FUNCTION_BLOCK TM_DO32 (* Composite Function Block Type *)
  (* Standard: 61499-2 *)
  (* Version 0.0, 21/08/2026, template *)
  PACKAGE Hidryco.HidrycoLib;
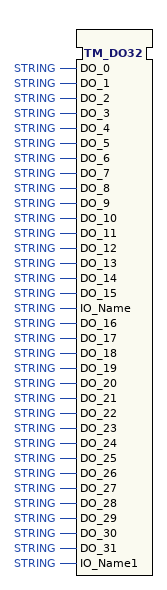
  VAR_INPUT
    DO_0 : STRING;
    DO_1 : STRING;
    DO_2 : STRING;
    DO_3 : STRING;
    DO_4 : STRING;
    DO_5 : STRING;
    DO_6 : STRING;
    DO_7 : STRING;
    DO_8 : STRING;
    DO_9 : STRING;
    DO_10 : STRING;
    DO_11 : STRING;
    DO_12 : STRING;
    DO_13 : STRING;
    DO_14 : STRING;
    DO_15 : STRING;
    IO_Name : STRING;
    DO_16 : STRING;
    DO_17 : STRING;
    DO_18 : STRING;
    DO_19 : STRING;
    DO_20 : STRING;
    DO_21 : STRING;
    DO_22 : STRING;
    DO_23 : STRING;
    DO_24 : STRING;
    DO_25 : STRING;
    DO_26 : STRING;
    DO_27 : STRING;
    DO_28 : STRING;
    DO_29 : STRING;
    DO_30 : STRING;
    DO_31 : STRING;
    IO_Name1 : STRING;
  END_VAR
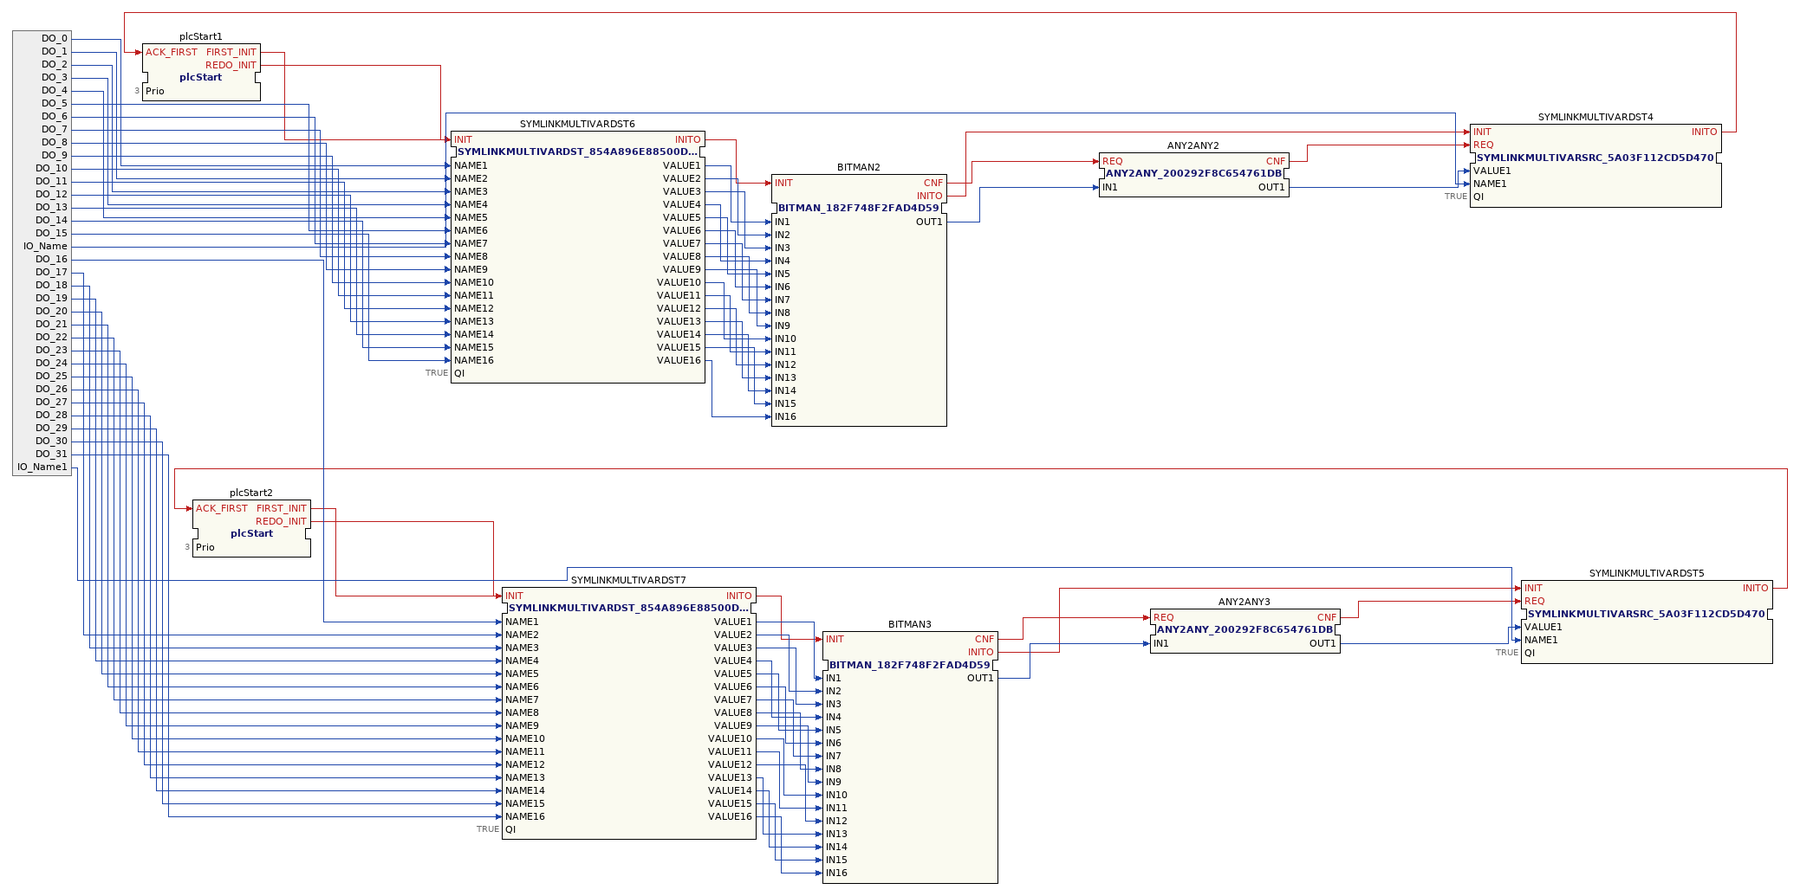
  FBS
    BITMAN2 : BITMAN_182F748F2FAD4D59; {SET_ATTRIBUTE(Configuration.GenericFBType.InterfaceParams, Runtime.Standard#CNTIN:=16;CNTOUT:=1;IN${CNTIN$}:BOOL,BOOL,BOOL,BOOL,BOOL,BOOL,BOOL,BOOL,BOOL,BOOL,BOOL,BOOL,BOOL,BOOL,BOOL,BOOL;OUT${CNTOUT$}:WORD)}
    ANY2ANY2 : ANY2ANY_200292F8C654761DB; {SET_ATTRIBUTE(Configuration.GenericFBType.InterfaceParams, Runtime.Standard#CNT:=1;IN${CNT$}:WORD;OUT${CNT$}:INT)}
    SYMLINKMULTIVARDST4 : SYMLINKMULTIVARSRC_5A03F112CD5D470(QI := TRUE); {SET_ATTRIBUTE(Configuration.GenericFBType.InterfaceParams, Runtime.System#I:=1;VALUE${I$}:INT)}
    SYMLINKMULTIVARDST6 : SYMLINKMULTIVARDST_854A896E88500D19(QI := TRUE); {SET_ATTRIBUTE(Configuration.GenericFBType.InterfaceParams, Runtime.System#I:=16;VALUE${I$}:BOOL,BOOL,BOOL,BOOL,BOOL,BOOL,BOOL,BOOL,BOOL,BOOL,BOOL,BOOL,BOOL,BOOL,BOOL,BOOL)}
    plcStart1 : plcStart(Prio := 3);
    BITMAN3 : BITMAN_182F748F2FAD4D59; {SET_ATTRIBUTE(Configuration.GenericFBType.InterfaceParams, Runtime.Standard#CNTIN:=16;CNTOUT:=1;IN${CNTIN$}:BOOL,BOOL,BOOL,BOOL,BOOL,BOOL,BOOL,BOOL,BOOL,BOOL,BOOL,BOOL,BOOL,BOOL,BOOL,BOOL;OUT${CNTOUT$}:WORD)}
    ANY2ANY3 : ANY2ANY_200292F8C654761DB; {SET_ATTRIBUTE(Configuration.GenericFBType.InterfaceParams, Runtime.Standard#CNT:=1;IN${CNT$}:WORD;OUT${CNT$}:INT)}
    SYMLINKMULTIVARDST5 : SYMLINKMULTIVARSRC_5A03F112CD5D470(QI := TRUE); {SET_ATTRIBUTE(Configuration.GenericFBType.InterfaceParams, Runtime.System#I:=1;VALUE${I$}:INT)}
    SYMLINKMULTIVARDST7 : SYMLINKMULTIVARDST_854A896E88500D19(QI := TRUE); {SET_ATTRIBUTE(Configuration.GenericFBType.InterfaceParams, Runtime.System#I:=16;VALUE${I$}:BOOL,BOOL,BOOL,BOOL,BOOL,BOOL,BOOL,BOOL,BOOL,BOOL,BOOL,BOOL,BOOL,BOOL,BOOL,BOOL)}
    plcStart2 : plcStart(Prio := 3);
  END_FBS
  EVENT_CONNECTIONS
    BITMAN2.CNF TO ANY2ANY2.REQ;
    BITMAN2.INITO TO SYMLINKMULTIVARDST4.INIT;
    ANY2ANY2.CNF TO SYMLINKMULTIVARDST4.REQ;
    SYMLINKMULTIVARDST6.INITO TO BITMAN2.INIT;
    plcStart1.FIRST_INIT TO SYMLINKMULTIVARDST6.INIT;
    plcStart1.REDO_INIT TO SYMLINKMULTIVARDST6.INIT;
    SYMLINKMULTIVARDST4.INITO TO plcStart1.ACK_FIRST;
    BITMAN3.CNF TO ANY2ANY3.REQ;
    BITMAN3.INITO TO SYMLINKMULTIVARDST5.INIT;
    ANY2ANY3.CNF TO SYMLINKMULTIVARDST5.REQ;
    SYMLINKMULTIVARDST7.INITO TO BITMAN3.INIT;
    plcStart2.FIRST_INIT TO SYMLINKMULTIVARDST7.INIT;
    plcStart2.REDO_INIT TO SYMLINKMULTIVARDST7.INIT;
    SYMLINKMULTIVARDST5.INITO TO plcStart2.ACK_FIRST;
  END_CONNECTIONS
  DATA_CONNECTIONS
    BITMAN2.OUT1 TO ANY2ANY2.IN1;
    ANY2ANY2.OUT1 TO SYMLINKMULTIVARDST4.VALUE1;
    SYMLINKMULTIVARDST6.VALUE1 TO BITMAN2.IN1;
    SYMLINKMULTIVARDST6.VALUE2 TO BITMAN2.IN2;
    SYMLINKMULTIVARDST6.VALUE3 TO BITMAN2.IN3;
    SYMLINKMULTIVARDST6.VALUE4 TO BITMAN2.IN4;
    SYMLINKMULTIVARDST6.VALUE5 TO BITMAN2.IN5;
    SYMLINKMULTIVARDST6.VALUE6 TO BITMAN2.IN6;
    SYMLINKMULTIVARDST6.VALUE7 TO BITMAN2.IN7;
    SYMLINKMULTIVARDST6.VALUE8 TO BITMAN2.IN8;
    SYMLINKMULTIVARDST6.VALUE9 TO BITMAN2.IN9;
    SYMLINKMULTIVARDST6.VALUE10 TO BITMAN2.IN10;
    SYMLINKMULTIVARDST6.VALUE11 TO BITMAN2.IN11;
    SYMLINKMULTIVARDST6.VALUE12 TO BITMAN2.IN12;
    SYMLINKMULTIVARDST6.VALUE13 TO BITMAN2.IN13;
    SYMLINKMULTIVARDST6.VALUE14 TO BITMAN2.IN14;
    SYMLINKMULTIVARDST6.VALUE15 TO BITMAN2.IN15;
    SYMLINKMULTIVARDST6.VALUE16 TO BITMAN2.IN16;
    DO_0 TO SYMLINKMULTIVARDST6.NAME1;
    DO_1 TO SYMLINKMULTIVARDST6.NAME2;
    DO_2 TO SYMLINKMULTIVARDST6.NAME3;
    DO_3 TO SYMLINKMULTIVARDST6.NAME4;
    DO_4 TO SYMLINKMULTIVARDST6.NAME5;
    DO_5 TO SYMLINKMULTIVARDST6.NAME6;
    DO_6 TO SYMLINKMULTIVARDST6.NAME7;
    DO_7 TO SYMLINKMULTIVARDST6.NAME8;
    DO_8 TO SYMLINKMULTIVARDST6.NAME9;
    DO_9 TO SYMLINKMULTIVARDST6.NAME10;
    DO_10 TO SYMLINKMULTIVARDST6.NAME11;
    DO_11 TO SYMLINKMULTIVARDST6.NAME12;
    DO_12 TO SYMLINKMULTIVARDST6.NAME13;
    DO_13 TO SYMLINKMULTIVARDST6.NAME14;
    DO_14 TO SYMLINKMULTIVARDST6.NAME15;
    DO_15 TO SYMLINKMULTIVARDST6.NAME16;
    IO_Name TO SYMLINKMULTIVARDST4.NAME1;
    BITMAN3.OUT1 TO ANY2ANY3.IN1;
    ANY2ANY3.OUT1 TO SYMLINKMULTIVARDST5.VALUE1;
    SYMLINKMULTIVARDST7.VALUE1 TO BITMAN3.IN1;
    SYMLINKMULTIVARDST7.VALUE2 TO BITMAN3.IN2;
    SYMLINKMULTIVARDST7.VALUE3 TO BITMAN3.IN3;
    SYMLINKMULTIVARDST7.VALUE4 TO BITMAN3.IN4;
    SYMLINKMULTIVARDST7.VALUE5 TO BITMAN3.IN5;
    SYMLINKMULTIVARDST7.VALUE6 TO BITMAN3.IN6;
    SYMLINKMULTIVARDST7.VALUE7 TO BITMAN3.IN7;
    SYMLINKMULTIVARDST7.VALUE8 TO BITMAN3.IN8;
    SYMLINKMULTIVARDST7.VALUE9 TO BITMAN3.IN9;
    SYMLINKMULTIVARDST7.VALUE10 TO BITMAN3.IN10;
    SYMLINKMULTIVARDST7.VALUE11 TO BITMAN3.IN11;
    SYMLINKMULTIVARDST7.VALUE12 TO BITMAN3.IN12;
    SYMLINKMULTIVARDST7.VALUE13 TO BITMAN3.IN13;
    SYMLINKMULTIVARDST7.VALUE14 TO BITMAN3.IN14;
    SYMLINKMULTIVARDST7.VALUE15 TO BITMAN3.IN15;
    SYMLINKMULTIVARDST7.VALUE16 TO BITMAN3.IN16;
    DO_16 TO SYMLINKMULTIVARDST7.NAME1;
    DO_17 TO SYMLINKMULTIVARDST7.NAME2;
    DO_18 TO SYMLINKMULTIVARDST7.NAME3;
    DO_19 TO SYMLINKMULTIVARDST7.NAME4;
    DO_20 TO SYMLINKMULTIVARDST7.NAME5;
    DO_21 TO SYMLINKMULTIVARDST7.NAME6;
    DO_22 TO SYMLINKMULTIVARDST7.NAME7;
    DO_23 TO SYMLINKMULTIVARDST7.NAME8;
    DO_24 TO SYMLINKMULTIVARDST7.NAME9;
    DO_25 TO SYMLINKMULTIVARDST7.NAME10;
    DO_26 TO SYMLINKMULTIVARDST7.NAME11;
    DO_27 TO SYMLINKMULTIVARDST7.NAME12;
    DO_28 TO SYMLINKMULTIVARDST7.NAME13;
    DO_29 TO SYMLINKMULTIVARDST7.NAME14;
    DO_30 TO SYMLINKMULTIVARDST7.NAME15;
    DO_31 TO SYMLINKMULTIVARDST7.NAME16;
    IO_Name1 TO SYMLINKMULTIVARDST5.NAME1;
  END_CONNECTIONS
END_FUNCTION_BLOCK
